Yaskawa INFORM job: LTEDSRCH.JBI

/JOB
//NAME LTEDSRCH
//POS
///NPOS 0,0,0,0,0,0
//INST
///DATE 2019/11/18 20:46
///ATTR SC,RW,MC
///GROUP1 RB1,BS1
///LVARS 2,0,0,0,0,0,0,0
NOP
GETARG LB000 IARG#(1)
GETARG LB001 IARG#(2)
JUMP *END IF LB000<>1
SKILLSND ATTR=3 "LSRCHED LT:1"
*END
END
